Universal Robots PolyScope program: Lab_exe_8_1_140.urp

Program Lab_exe_8_1_140 (createdIn=3.2.19293 lastSavedIn=3.2.19293 directory=/programs installation=default robotSerialNumber=2015351391)
Calibrated DH parameters: a=[0.000352, -0.161198, -0.373486, 0.00005, 0.000049, 0]; d=[0.089268, 352.477598, -320.08558, -32.281492, 0.094939, 0.082518]; alpha=[1.570728, 0.001116, -0.003686, 1.571189, -1.570572, 0]; deltaTheta=[-0.000012, 1.181849, -1.491165, 0.309495, -0.000007, 0.000025]
Robot Program (runOnlyOnce=false motionType=MoveJ speed=1.047198 acceleration=1.396263 recalculateMotions=false)
  Pallet pattern(dimensionality=Square firstAxisCount=7 secondAxisCount=4 thirdAxisCount=5 motionType=MoveL speed=0.25 acceleration=1.2 recalculateMotions=false, counterVariable(name=cnt_1, initializeExpression=0), patternPoseVariable(name=位姿_1), feature=Base, children(Waypoint(type=Fixed name=a1st_Corner_1, position(joints=2.582643141693131, -2.088075508146252, -1.9571173579004864, -0.6673388236395041, 1.5690286006888252, 4.149548872293666 pose=-0.40525447916334395, 0.3849287182929952, 0.06805445183381634, -1.6716414602742922E-4, -3.141439672903999, -1.3355598048384883E-4), poseInFeatureCoordinates=[-0.405254, 0.384929, 0.068054, -0.000167, -3.14144, -0.000134], outputFlangePose=[-0.405292, 0.384877, 0.068069, -0.000133, -3.141303, -0.000034]), Waypoint(type=Fixed name=a2nd_Corner_1, position(joints=2.238721458097343, -2.5440105504774913, -1.0677191189711417, -1.1008640332903532, 1.5682333964263835, 3.8062756161575844 pose=-0.4052688246082992, 0.6940130736959474, 0.06805805429031908, -1.4583686165772024E-4, -3.14150622024288, 6.0000958538445606E-5), poseInFeatureCoordinates=[-0.405269, 0.694013, 0.068058, -0.000146, -3.141506, 0.00006], outputFlangePose=[-0.405292, 0.694027, 0.068069, -0.000133, -3.141303, -0.000034]), Waypoint(type=Fixed name=a3rd_Corner_1, position(joints=2.010509916984664, -2.343507132312279, -1.441440890381032, -0.9276987373055441, 1.5685450851040228, 3.57771898942143 pose=-0.19932441854465685, 0.6857466752949721, 0.07568574548320177, -1.2693840113585825E-4, -3.141322916060241, 6.672113611315508E-5), poseInFeatureCoordinates=[-0.199324, 0.685747, 0.075686, -0.000127, -3.141323, 0.000067], outputFlangePose=[-0.199308, 0.68574, 0.0757, -0.000133, -3.141303, -0.000034]), Waypoint(type=Fixed name=a4th_Corner_1, position(joints=2.313424045091331, -1.8880399911078403, -2.323065954819384, -0.5014713964448845, 1.5695189914280527, 3.8803182886818175 pose=-0.19928480595341969, 0.38161911331091786, 0.0666825185953147, -1.2763845206907473E-4, -3.1415178813605036, -6.643162239517727E-5), poseInFeatureCoordinates=[-0.199285, 0.381619, 0.066683, -0.000128, -3.141518, -0.000066], outputFlangePose=[-0.199308, 0.381597, 0.06667, -0.000133, -3.141303, -0.000034]))); actionSequence(name=托盘序列 motionType=MoveL speed=0.25 acceleration=1.2 recalculateMotions=false, anchorWaypoint(type=Fixed name=模式点_1, position(joints=2.582643141693131, -2.088075508146252, -1.9571173579004864, -0.6673388236395041, 1.5690286006888252, 4.149548872293666 pose=-0.4053089109546333, 0.3849151819327164, 0.06809603996897211, -9.182204698629077E-5, -3.1412904149525724, -2.5885630344950675E-4), poseInFeatureCoordinates=[-0.405309, 0.384915, 0.068096, -0.000092, -3.14129, -0.000259], outputFlangePose=[-0.405292, 0.384877, 0.068069, -0.000133, -3.141303, -0.000034]), feature=Base, children(Waypoint(type=Fixed name=方式_1, position(joints=2.582595376657776, -1.9258952385460368, -1.8952388111768412, -0.8913968349047998, 1.5681608593537268, 4.149996907722099 pose=-0.40530293419349106, 0.3848843934638523, 0.1586936979858413, -2.3611149661249454E-4, -3.1412609243015774, -2.1404800871644547E-4), poseInFeatureCoordinates=[-0.405303, 0.384884, 0.158694, -0.000236, -3.141261, -0.000214], outputFlangePose=[-0.405292, 0.384877, 0.158684, -0.000133, -3.141303, -0.000034]), Waypoint=模式点_1, Set(type=DigitalOutput, pin=Lamp, digitalValue=1), Wait(type=Sleep, waitTime=0.5), Waypoint(type=Fixed name=退出_1, position(joints=2.582595376657776, -1.9258952385460368, -1.8952388111768412, -0.8913968349047998, 1.5681608593537268, 4.149996907722099 pose=-0.40530370199502896, 0.38486306114392277, 0.1586723605399197, -1.223834237907333E-4, -3.141326202067636, 1.1772033102516707E-4), poseInFeatureCoordinates=[-0.405304, 0.384863, 0.158672, -0.000122, -3.141326, 0.000118], outputFlangePose=[-0.405292, 0.384877, 0.158684, -0.000133, -3.141303, -0.000034])))
    Pattern -> pattern
    AnchoredSequence -> 托盘序列
